LIN {X 0,Y 21.95,Z 458.517,A -85,B 0,C 180,E1 -31714.406,E2 -31714.406} C_VEL
LIN {X 0,Y 18.669,Z 455.649,A -85,B 0,C 180,E1 -31732.501,E2 -31732.501} C_VEL
LIN {X 0,Y 17.592,Z 454.28,A -85,B 0,C 180,E1 -31738.229,E2 -31738.229} C_VEL
LIN {X 0,Y 14.214,Z 449.35,A -85,B 0,C 180,E1 -31755.672,E2 -31755.672} C_VEL
LIN {X 0,Y 10.98,Z 441.099,A -85,B 0,C 180,E1 -31788.665,E2 -31788.665} C_VEL
LIN {X 0,Y 12.349,Z 431.094,A -85,B 0,C 180,E1 -31827.539,E2 -31827.539} C_VEL
LIN {X 0,Y 17.38,Z 418.57,A -85,B 0,C 180,E1 -31851.795,E2 -31851.795} C_VEL
LIN {X 0,Y 19,Z 414.708,A -85,B 0,C 180,E1 -31856.022,E2 -31856.022} C_VEL
LIN {X 0,Y 19.089,Z 413.104,A -85,B 0,C 180,E1 -31859.999,E2 -31859.999} C_VEL
LIN {X 0,Y 18.959,Z 411.089,A -85,B 0,C 180,E1 -31866.564,E2 -31866.564} C_VEL
LIN {X 0,Y 18.463,Z 410.665,A -85,B 0,C 180,E1 -31871.072,E2 -31871.072} C_VEL
LIN {X 0,Y 17.071,Z 411.616,A -85,B 0,C 180,E1 -31878.8,E2 -31878.8} C_VEL
LIN {X 0,Y 14.464,Z 415.233,A -85,B 0,C 180,E1 -31897.157,E2 -31897.157} C_VEL
LIN {X 0,Y 14.345,Z 415.691,A -85,B 0,C 180,E1 -31904.038,E2 -31904.038} C_VEL
LIN {X 0,Y 14.536,Z 415.828,A -85,B 0,C 180,E1 -31909.54,E2 -31909.54} C_VEL
LIN {X 0,Y 14.608,Z 416.494,A -85,B 0,C 180,E1 -31915.709,E2 -31915.709} C_VEL
LIN {X 0,Y 13.138,Z 421.53,A -85,B 0,C 180,E1 -31931.207,E2 -31931.207} C_VEL
LIN {X 0,Y 10.012,Z 426.431,A -85,B 0,C 180,E1 -31937.224,E2 -31937.224} C_VEL
LIN {X 0,Y 3.068,Z 438.022,A -85,B 0,C 180,E1 -32007.256,E2 -32007.256} C_VEL
LIN {X 0,Y 10.186,Z 448.082,A -85,B 0,C 180,E1 -32083.628,E2 -32083.628} C_VEL
LIN {X 0,Y 10.431,Z 448.25,A -85,B 0,C 180,E1 -32087.643,E2 -32087.643} C_VEL
LIN {X 0,Y 4.309,Z 439.995,A -85,B 0,C 180,E1 -32130,E2 -32130} C_VEL
LIN {X 0,Y 7.039,Z 429.717,A -85,B 0,C 180,E1 -32216.746,E2 -32216.746} C_VEL
LIN {X 0,Y 13.719,Z 418.196,A -85,B 0,C 180,E1 -32234.396,E2 -32234.396} C_VEL
LIN {X 0,Y 14.591,Z 416.6,A -85,B 0,C 180,E1 -32235.562,E2 -32235.562} C_VEL
LIN {X 0,Y 14.88,Z 415.575,A -85,B 0,C 180,E1 -32239.159,E2 -32239.159} C_VEL
LIN {X 0,Y 14.508,Z 415.32,A -85,B 0,C 180,E1 -32248.974,E2 -32248.974} C_VEL
LIN {X 0,Y 14.345,Z 415.691,A -85,B 0,C 180,E1 -32264.038,E2 -32264.038} C_VEL
LIN {X 0,Y 14.616,Z 417.681,A -85,B 0,C 180,E1 -32271.103,E2 -32271.103} C_VEL
LIN {X 0,Y 14.616,Z 600,A -85,B 0,C 180,E1 -32271.103,E2 -32271.103} C_VEL
LIN {X 0,Y 14.616,Z 600,A -85,B 0,C 180,E1 -32271.103,E2 -32271.103}

QRS_NEXT_CUT()

QRS_NEXT()
QRS_HOME()

END
